PROGRAM LadderLogic_1
VAR
END_VAR
VAR // added by the converter: edge detectors and wires of the graphical bodies
    _w1, _w2, _w3 : BOOL;
END_VAR

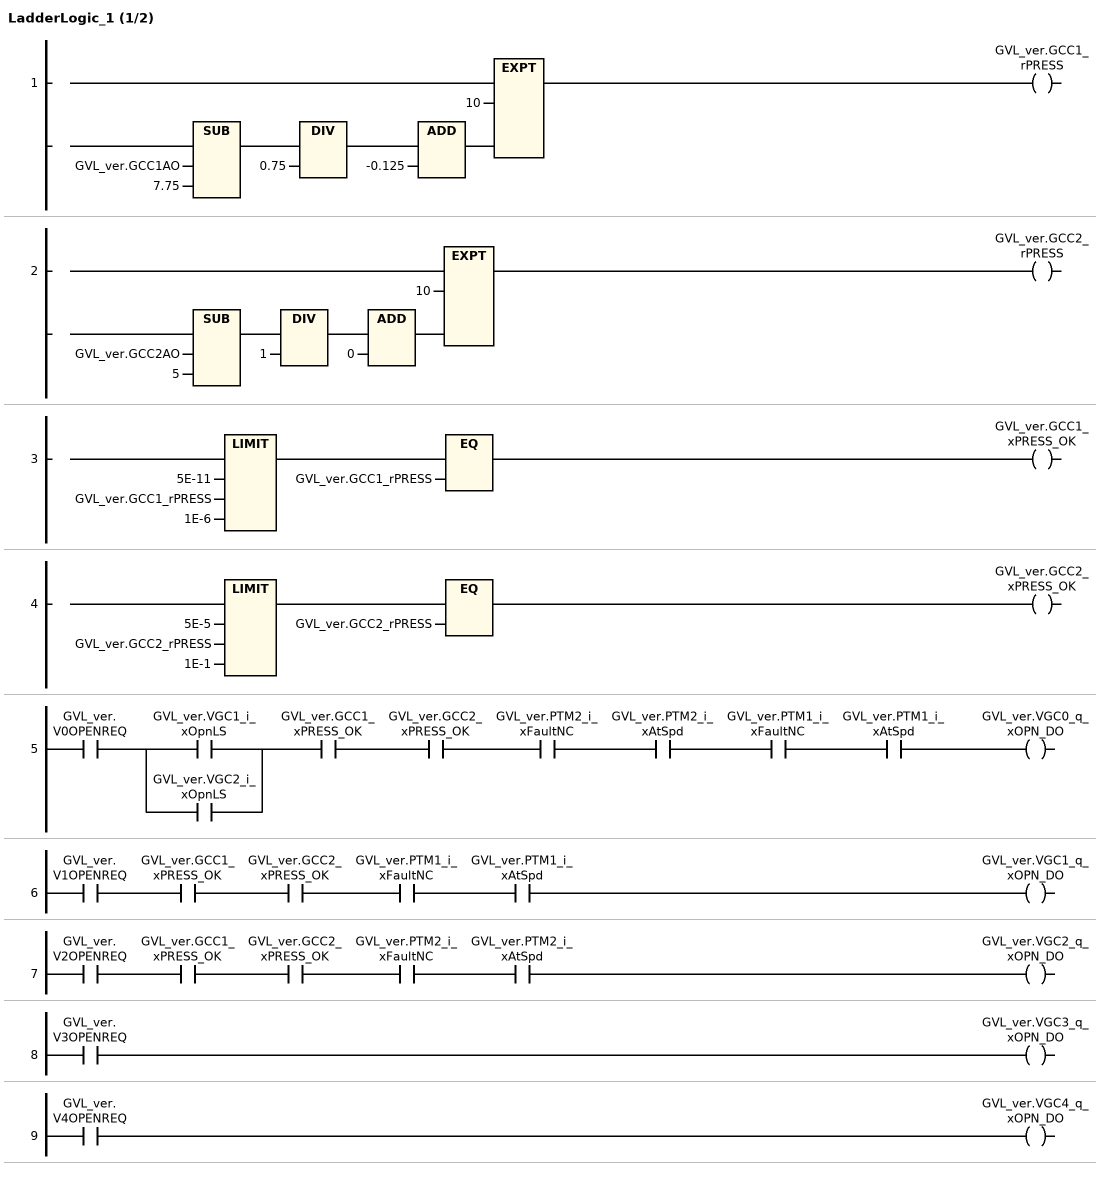
// NETWORK 1
GVL_ver.GCC1_rPRESS := EXPT(10, (GVL_ver.GCC1AO - 7.75) / 0.75 + -0.125);

// NETWORK 2
GVL_ver.GCC2_rPRESS := EXPT(10, (GVL_ver.GCC2AO - 5) / 1 + 0);

// NETWORK 3
GVL_ver.GCC1_xPRESS_OK := LIMIT(5E-11, GVL_ver.GCC1_rPRESS, 1E-6) = GVL_ver.GCC1_rPRESS;

// NETWORK 4
GVL_ver.GCC2_xPRESS_OK := LIMIT(5E-5, GVL_ver.GCC2_rPRESS, 1E-1) = GVL_ver.GCC2_rPRESS;

// NETWORK 5
GVL_ver.VGC0_q_xOPN_DO := GVL_ver.V0OPENREQ AND (GVL_ver.VGC1_i_xOpnLS OR GVL_ver.VGC2_i_xOpnLS) AND GVL_ver.GCC1_xPRESS_OK AND GVL_ver.GCC2_xPRESS_OK AND GVL_ver.PTM2_i_xFaultNC AND GVL_ver.PTM2_i_xAtSpd AND GVL_ver.PTM1_i_xFaultNC AND GVL_ver.PTM1_i_xAtSpd;

// NETWORK 6
GVL_ver.VGC1_q_xOPN_DO := GVL_ver.V1OPENREQ AND GVL_ver.GCC1_xPRESS_OK AND GVL_ver.GCC2_xPRESS_OK AND GVL_ver.PTM1_i_xFaultNC AND GVL_ver.PTM1_i_xAtSpd;

// NETWORK 7
GVL_ver.VGC2_q_xOPN_DO := GVL_ver.V2OPENREQ AND GVL_ver.GCC1_xPRESS_OK AND GVL_ver.GCC2_xPRESS_OK AND GVL_ver.PTM2_i_xFaultNC AND GVL_ver.PTM2_i_xAtSpd;

// NETWORK 8
GVL_ver.VGC3_q_xOPN_DO := GVL_ver.V3OPENREQ;

// NETWORK 9
GVL_ver.VGC4_q_xOPN_DO := GVL_ver.V4OPENREQ;

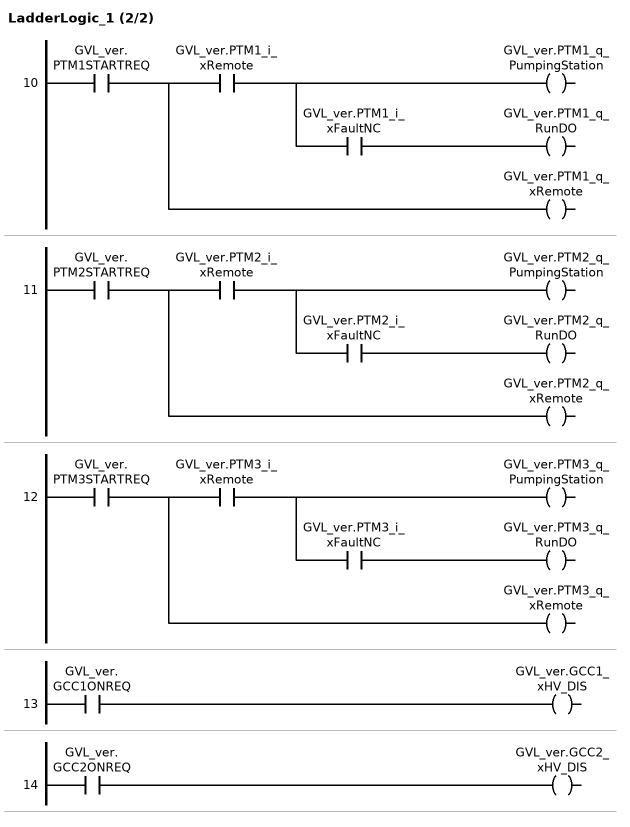
// NETWORK 10
_w1 := GVL_ver.PTM1STARTREQ AND GVL_ver.PTM1_i_xRemote;
GVL_ver.PTM1_q_PumpingStation := _w1;
GVL_ver.PTM1_q_RunDO := _w1 AND GVL_ver.PTM1_i_xFaultNC;
GVL_ver.PTM1_q_xRemote := GVL_ver.PTM1STARTREQ;

// NETWORK 11
_w2 := GVL_ver.PTM2STARTREQ AND GVL_ver.PTM2_i_xRemote;
GVL_ver.PTM2_q_PumpingStation := _w2;
GVL_ver.PTM2_q_RunDO := _w2 AND GVL_ver.PTM2_i_xFaultNC;
GVL_ver.PTM2_q_xRemote := GVL_ver.PTM2STARTREQ;

// NETWORK 12
_w3 := GVL_ver.PTM3STARTREQ AND GVL_ver.PTM3_i_xRemote;
GVL_ver.PTM3_q_PumpingStation := _w3;
GVL_ver.PTM3_q_RunDO := _w3 AND GVL_ver.PTM3_i_xFaultNC;
GVL_ver.PTM3_q_xRemote := GVL_ver.PTM3STARTREQ;

// NETWORK 13
GVL_ver.GCC1_xHV_DIS := GVL_ver.GCC1ONREQ;

// NETWORK 14
GVL_ver.GCC2_xHV_DIS := GVL_ver.GCC2ONREQ;

END_PROGRAM

(* stored: Version 1.1.0.1, ProductVersion 3.1.4022.3
   POU LadderLogic_1: Id {cced6ceb-cd51-44d1-b841-27d4ac87152c}, SpecialFunc None *)
